TYPE ST_DI_StandardChannel :
STRUCT
	Status : INT;
	Value : INT;
END_STRUCT
END_TYPE

(* stored: Version 1.1.0.1, ProductVersion 3.1.4024.11
   DUT ST_DI_StandardChannel: Id {9b74c086-4b23-476a-88ba-5b66409ee090} *)
